PROGRAM TestfbSoEWrite
VAR
	fbSoEWrite : FB_SoEWrite;
	nTorqueLimit : UINT := 980;
	
	bExecute : BOOL;
	stFeedbackOneType : ST_FeedbackOneType;
END_VAR


stFeedbackOneType.Manufacturer := E_Manufacturer.Hengstler;

fbSoEWrite(
	Axis:= Motion.Axis1, 
	NetId:= '10.100.6.93.1.1', 
	Idn:= S_0_IDNs+150, 
	Element:= 16#40, 
	pSrcBuf:= ADR(stFeedbackOneType), 
	BufLen:= SIZEOF(stFeedbackOneType), 
	Execute:= bExecute, 
	Timeout:= , 
	Password:= , 
	Busy=> , 
	Error=> , 
	AdsErrId=> , 
	SercosErrId=> );

END_PROGRAM

(* stored: Version 1.1.0.1, ProductVersion 3.1.4024.12
   POU TestfbSoEWrite: Id {1fe0071d-fd39-4fc0-896e-8231765b6dc1}, SpecialFunc None *)
